{attribute addProperty BoxType "EL3632-0000-0016"}
{attribute addProperty Id "Ch2_ValueAT %I*INT162"}
{attribute addProperty CRC "703390824"}
{attribute addProperty SizeInBites "16"}
{attribute addProperty SizeInBytes "2"}
TYPE Ch2_Sample_29ECE468 :
STRUCT
	{attribute addProperty Name "Ch2_Value"}
	Ch2_Value AT %I* : INT;
END_STRUCT
END_TYPE

(* stored: Version 1.2.0.0, ProductVersion 3.1.4024.9
   DUT Ch2_Sample_29ECE468: Id {24c0ffde-8083-463a-8501-c4e1c8618e22} *)
